// This function has been automatically generated from the project information.
{attribute 'signature_flag' := '1073741824'}
{attribute 'TcGenerated'}
{attribute 'no-analysis'}
FUNCTION F_GetCompany : WSTRING
VAR_INPUT
	
END_VAR

F_GetCompany := "Simmel";

END_FUNCTION

(* stored: Version 1.1.0.1
   POU F_GetCompany: Id {e5cdeab6-d1cc-46bd-aaec-7d4fd99da541}, SpecialFunc None *)
